{attribute 'linkalways'} 
{attribute 'no_explicit_call' := 'This FB is a CLASS and must be accessed using methods or properties'}
{attribute 'enable_dynamic_creation'}
FUNCTION_BLOCK PUBLIC DeserializationFailedNodeNotSupportedAlarm EXTENDS Alarm
VAR
	state : (CLEARED, RAISED);
	_reason : T_MAXSTRING;
END_VAR

PROPERTY Active : BOOL
GET
Active := state <> CLEARED;
END_GET
END_PROPERTY

METHOD PUBLIC Clear
_reason := '';
state := CLEARED;
END_METHOD

PROPERTY PUBLIC Message : T_MaxString
GET
Message := 'Node type is not installed';
END_GET
END_PROPERTY

METHOD PUBLIC Raise
VAR_INPUT
	NodeType : T_MAXSTRING;
END_VAR
_reason := NodeType;
state := RAISED;
END_METHOD

PROPERTY Reason : T_MaxString
GET
Reason := _reason;
END_GET
END_PROPERTY

END_FUNCTION_BLOCK

(* stored: Version 1.1.0.1, ProductVersion 3.1.4024.12
   POU DeserializationFailedNodeNotSupportedAlarm: Id {8760a8c2-b7f4-42b1-8fb1-4e150dff7521}, SpecialFunc None
   Property Active: Id {ad045389-6112-456a-a667-a8dd25812b14}
   Get Get: Id {cef97d97-273a-4437-a51d-376b76ece23b}
   Method Clear: Id {7b2507cf-295d-4343-b7c8-3980a7008dbb}
   Property Message: Id {d3d07426-175b-4870-8778-2dbc984f06dd}
   Get Get: Id {07a4af6d-4bed-455e-a300-528f11c724b1}
   Method Raise: Id {d3655f05-8e18-4e49-8645-2500f3cd818a}
   Property Reason: Id {104dd125-7727-4097-9047-d795d8ce794b}
   Get Get: Id {caf1195d-8315-4795-9e55-3a7a0feba10d} *)
